(* Logix 5000 project; controller SX_V040001_C001 vendor 1 type 14 code 77 rev 16.22; software revision 16.04; part 33 of 35 *)
(* tags used below, declared in another part *)
   ALL_KINDS : INT[90];
   CMD : INT[36];
   EMPTYING : INT[18];
   G_DInput : DINT[3];
   loading : INT[19];
   METERING : INT[44];
   PARAMETER : INT[501];
   RECIPE_GENERAL : INT[405];
   REMOTE_DATA_IN : INT[510];
   REMOTE_DATA_OUT : INT[510];
   REMOTE_RECIPE : INT[405];
   REMOTE_SYSTEM : INT[38];
   RM_CMD : INT[9];
   s_bcc : INT;
   STATUS_SEND_PART_1 : INT[135];
   T_LIVEBIT_OFF : TIMER;
   T_LIVEBIT_ON : TIMER;
(* MainProgram, continued *)

ROUTINE RemoteComDeco_Direct   (* ladder *)
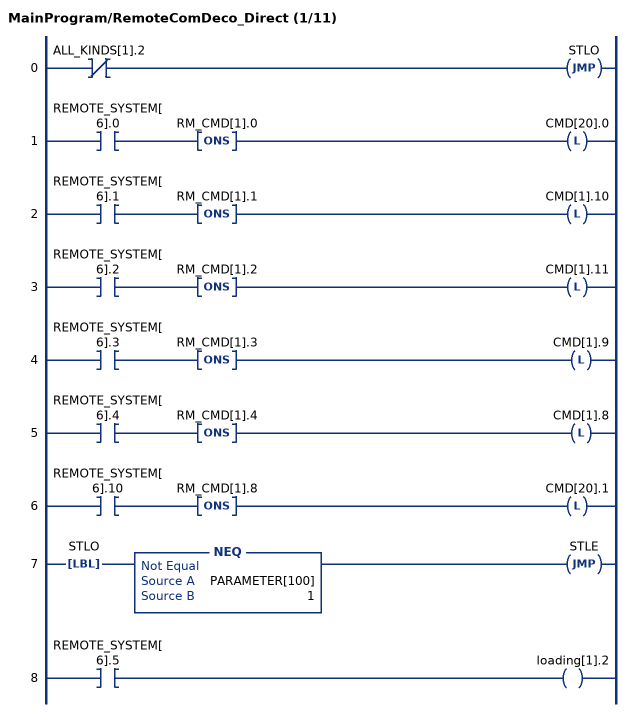
   0: XIO(ALL_KINDS[1].2)JMP(STLO);
   1: XIC(REMOTE_SYSTEM[6].0)ONS(RM_CMD[1].0)OTL(CMD[20].0);
   2: XIC(REMOTE_SYSTEM[6].1)ONS(RM_CMD[1].1)OTL(CMD[1].10);
   3: XIC(REMOTE_SYSTEM[6].2)ONS(RM_CMD[1].2)OTL(CMD[1].11);
   4: XIC(REMOTE_SYSTEM[6].3)ONS(RM_CMD[1].3)OTL(CMD[1].9);
   5: XIC(REMOTE_SYSTEM[6].4)ONS(RM_CMD[1].4)OTL(CMD[1].8);
   6: XIC(REMOTE_SYSTEM[6].10)ONS(RM_CMD[1].8)OTL(CMD[20].1);
   7: LBL(STLO)NEQ(PARAMETER[100],1)JMP(STLE);
   8: XIC(REMOTE_SYSTEM[6].5)OTE(loading[1].2);
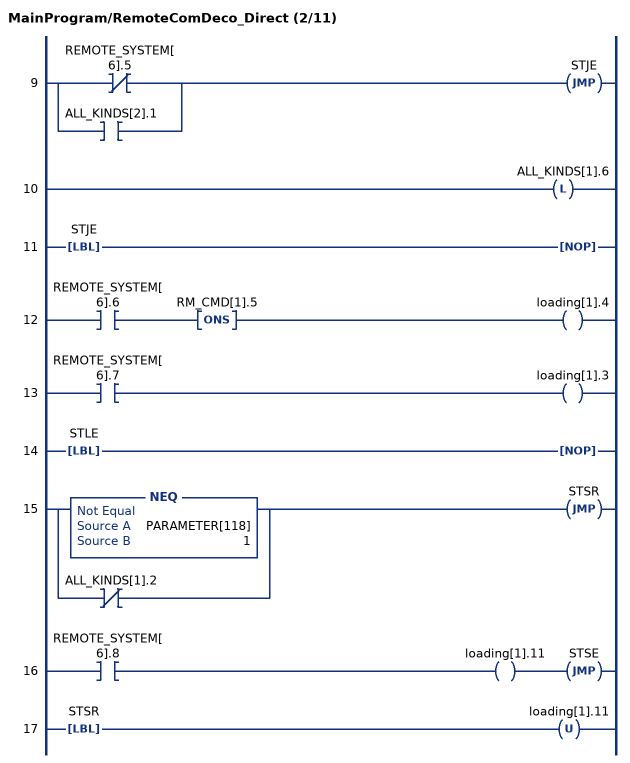
   9: [XIO(REMOTE_SYSTEM[6].5) ,XIC(ALL_KINDS[2].1) ]JMP(STJE);
   10: OTL(ALL_KINDS[1].6);
   11: LBL(STJE)NOP();
   12: XIC(REMOTE_SYSTEM[6].6)ONS(RM_CMD[1].5)OTE(loading[1].4);
   13: XIC(REMOTE_SYSTEM[6].7)OTE(loading[1].3);
   14: LBL(STLE)NOP();
   15: [NEQ(PARAMETER[118],1) ,XIO(ALL_KINDS[1].2) ]JMP(STSR);
   16: XIC(REMOTE_SYSTEM[6].8)OTE(loading[1].11)JMP(STSE);
   17: LBL(STSR)OTU(loading[1].11);
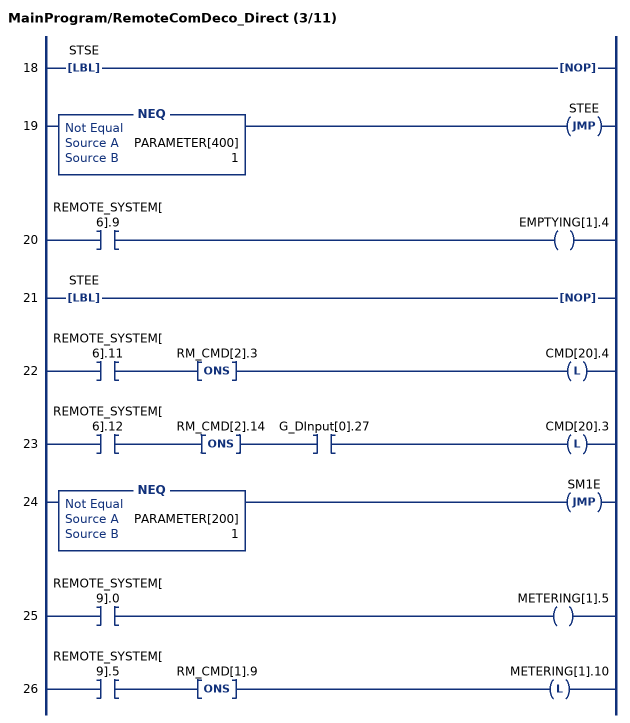
   18: LBL(STSE)NOP();
   19: NEQ(PARAMETER[400],1)JMP(STEE);
   20: XIC(REMOTE_SYSTEM[6].9)OTE(EMPTYING[1].4);
   21: LBL(STEE)NOP();
   22: XIC(REMOTE_SYSTEM[6].11)ONS(RM_CMD[2].3)OTL(CMD[20].4);
   23: XIC(REMOTE_SYSTEM[6].12)ONS(RM_CMD[2].14)XIC(G_DInput[0].27)OTL(CMD[20].3);
   24: NEQ(PARAMETER[200],1)JMP(SM1E);
   25: XIC(REMOTE_SYSTEM[9].0)OTE(METERING[1].5);
   26: XIC(REMOTE_SYSTEM[9].5)ONS(RM_CMD[1].9)OTL(METERING[1].10);
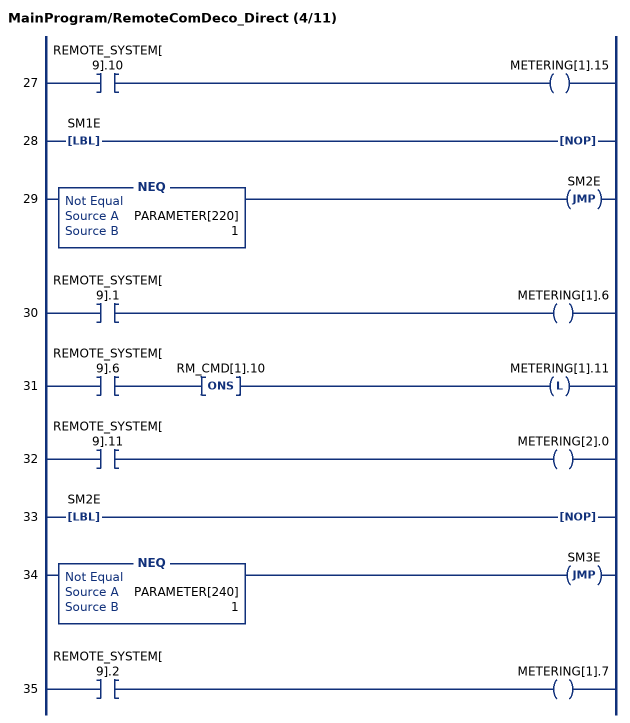
   27: XIC(REMOTE_SYSTEM[9].10)OTE(METERING[1].15);
   28: LBL(SM1E)NOP();
   29: NEQ(PARAMETER[220],1)JMP(SM2E);
   30: XIC(REMOTE_SYSTEM[9].1)OTE(METERING[1].6);
   31: XIC(REMOTE_SYSTEM[9].6)ONS(RM_CMD[1].10)OTL(METERING[1].11);
   32: XIC(REMOTE_SYSTEM[9].11)OTE(METERING[2].0);
   33: LBL(SM2E)NOP();
   34: NEQ(PARAMETER[240],1)JMP(SM3E);
   35: XIC(REMOTE_SYSTEM[9].2)OTE(METERING[1].7);
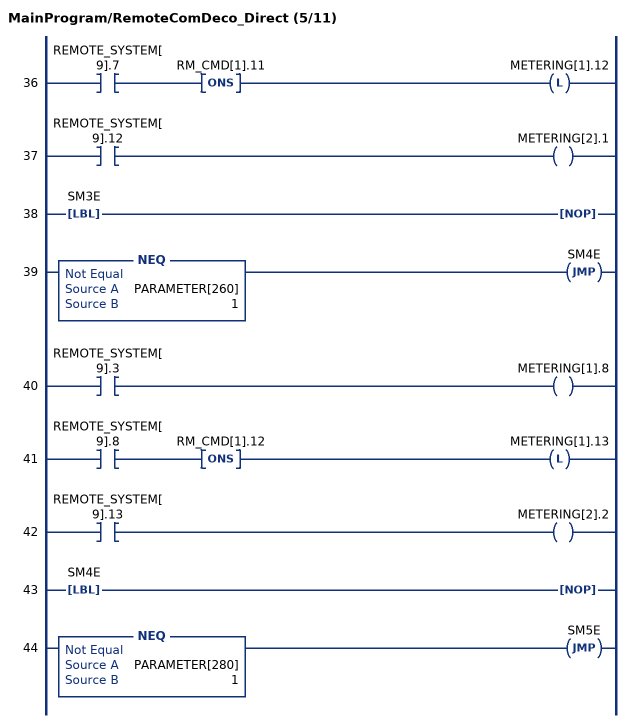
   36: XIC(REMOTE_SYSTEM[9].7)ONS(RM_CMD[1].11)OTL(METERING[1].12);
   37: XIC(REMOTE_SYSTEM[9].12)OTE(METERING[2].1);
   38: LBL(SM3E)NOP();
   39: NEQ(PARAMETER[260],1)JMP(SM4E);
   40: XIC(REMOTE_SYSTEM[9].3)OTE(METERING[1].8);
   41: XIC(REMOTE_SYSTEM[9].8)ONS(RM_CMD[1].12)OTL(METERING[1].13);
   42: XIC(REMOTE_SYSTEM[9].13)OTE(METERING[2].2);
   43: LBL(SM4E)NOP();
   44: NEQ(PARAMETER[280],1)JMP(SM5E);
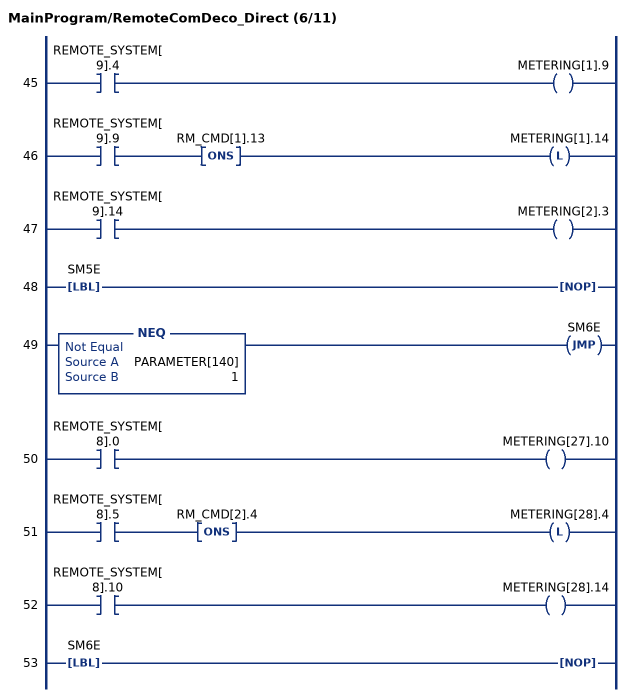
   45: XIC(REMOTE_SYSTEM[9].4)OTE(METERING[1].9);
   46: XIC(REMOTE_SYSTEM[9].9)ONS(RM_CMD[1].13)OTL(METERING[1].14);
   47: XIC(REMOTE_SYSTEM[9].14)OTE(METERING[2].3);
   48: LBL(SM5E)NOP();
   49: NEQ(PARAMETER[140],1)JMP(SM6E);
   50: XIC(REMOTE_SYSTEM[8].0)OTE(METERING[27].10);
   51: XIC(REMOTE_SYSTEM[8].5)ONS(RM_CMD[2].4)OTL(METERING[28].4);
   52: XIC(REMOTE_SYSTEM[8].10)OTE(METERING[28].14);
   53: LBL(SM6E)NOP();
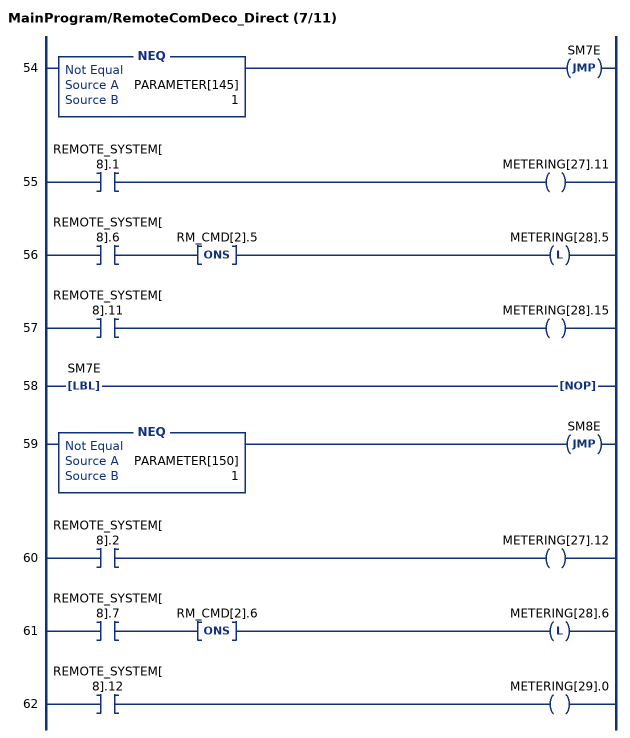
   54: NEQ(PARAMETER[145],1)JMP(SM7E);
   55: XIC(REMOTE_SYSTEM[8].1)OTE(METERING[27].11);
   56: XIC(REMOTE_SYSTEM[8].6)ONS(RM_CMD[2].5)OTL(METERING[28].5);
   57: XIC(REMOTE_SYSTEM[8].11)OTE(METERING[28].15);
   58: LBL(SM7E)NOP();
   59: NEQ(PARAMETER[150],1)JMP(SM8E);
   60: XIC(REMOTE_SYSTEM[8].2)OTE(METERING[27].12);
   61: XIC(REMOTE_SYSTEM[8].7)ONS(RM_CMD[2].6)OTL(METERING[28].6);
   62: XIC(REMOTE_SYSTEM[8].12)OTE(METERING[29].0);
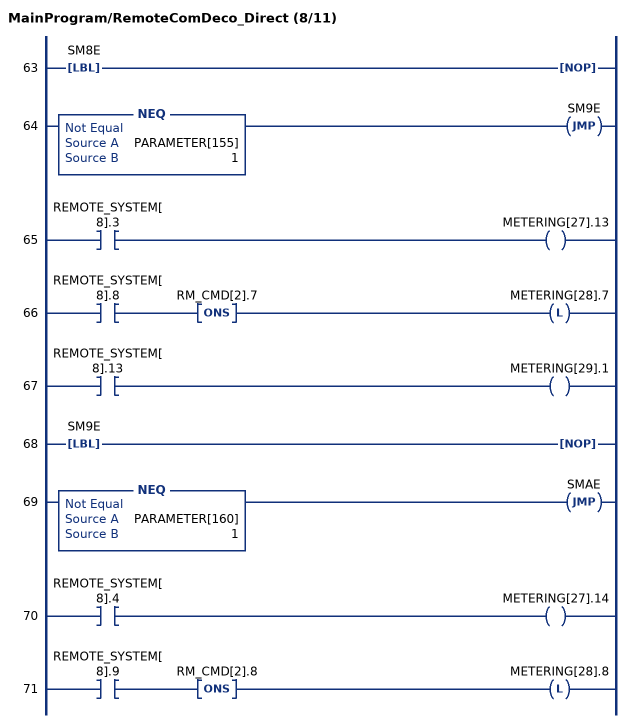
   63: LBL(SM8E)NOP();
   64: NEQ(PARAMETER[155],1)JMP(SM9E);
   65: XIC(REMOTE_SYSTEM[8].3)OTE(METERING[27].13);
   66: XIC(REMOTE_SYSTEM[8].8)ONS(RM_CMD[2].7)OTL(METERING[28].7);
   67: XIC(REMOTE_SYSTEM[8].13)OTE(METERING[29].1);
   68: LBL(SM9E)NOP();
   69: NEQ(PARAMETER[160],1)JMP(SMAE);
   70: XIC(REMOTE_SYSTEM[8].4)OTE(METERING[27].14);
   71: XIC(REMOTE_SYSTEM[8].9)ONS(RM_CMD[2].8)OTL(METERING[28].8);
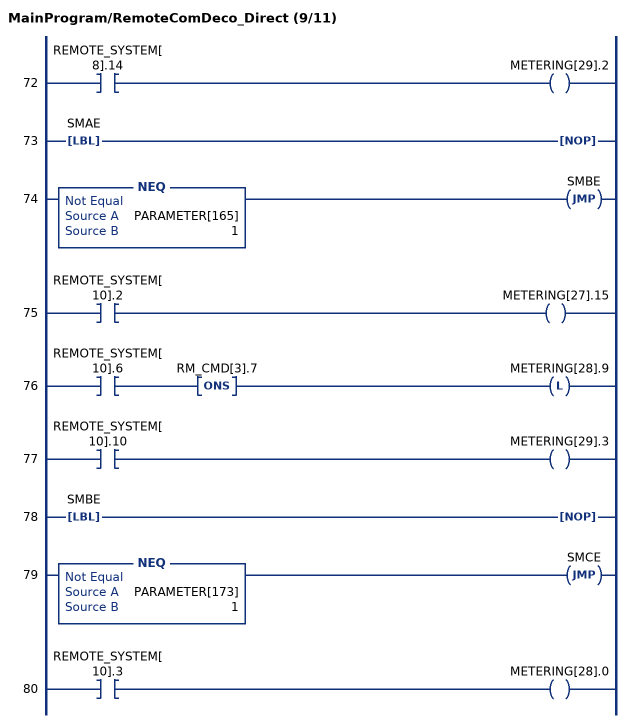
   72: XIC(REMOTE_SYSTEM[8].14)OTE(METERING[29].2);
   73: LBL(SMAE)NOP();
   74: NEQ(PARAMETER[165],1)JMP(SMBE);
   75: XIC(REMOTE_SYSTEM[10].2)OTE(METERING[27].15);
   76: XIC(REMOTE_SYSTEM[10].6)ONS(RM_CMD[3].7)OTL(METERING[28].9);
   77: XIC(REMOTE_SYSTEM[10].10)OTE(METERING[29].3);
   78: LBL(SMBE)NOP();
   79: NEQ(PARAMETER[173],1)JMP(SMCE);
   80: XIC(REMOTE_SYSTEM[10].3)OTE(METERING[28].0);
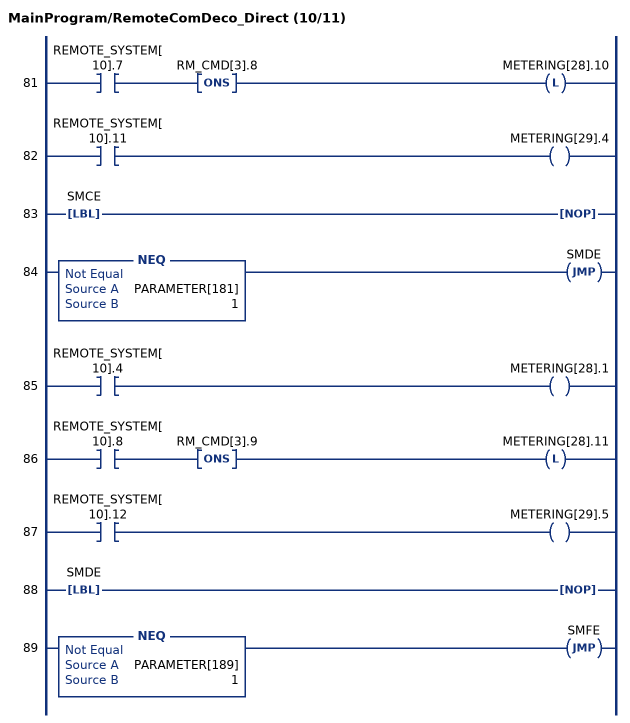
   81: XIC(REMOTE_SYSTEM[10].7)ONS(RM_CMD[3].8)OTL(METERING[28].10);
   82: XIC(REMOTE_SYSTEM[10].11)OTE(METERING[29].4);
   83: LBL(SMCE)NOP();
   84: NEQ(PARAMETER[181],1)JMP(SMDE);
   85: XIC(REMOTE_SYSTEM[10].4)OTE(METERING[28].1);
   86: XIC(REMOTE_SYSTEM[10].8)ONS(RM_CMD[3].9)OTL(METERING[28].11);
   87: XIC(REMOTE_SYSTEM[10].12)OTE(METERING[29].5);
   88: LBL(SMDE)NOP();
   89: NEQ(PARAMETER[189],1)JMP(SMFE);
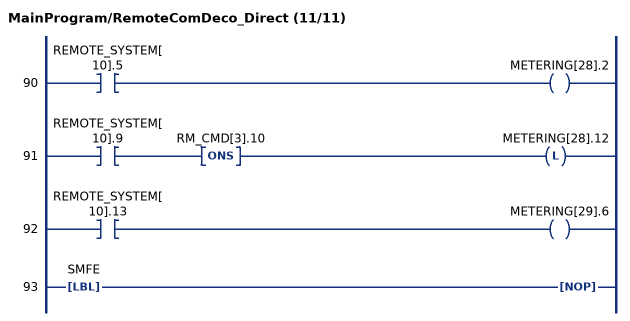
   90: XIC(REMOTE_SYSTEM[10].5)OTE(METERING[28].2);
   91: XIC(REMOTE_SYSTEM[10].9)ONS(RM_CMD[3].10)OTL(METERING[28].12);
   92: XIC(REMOTE_SYSTEM[10].13)OTE(METERING[29].6);
   93: LBL(SMFE)NOP();
END_ROUTINE

ROUTINE RemoteSystemHandler   (* ladder *)
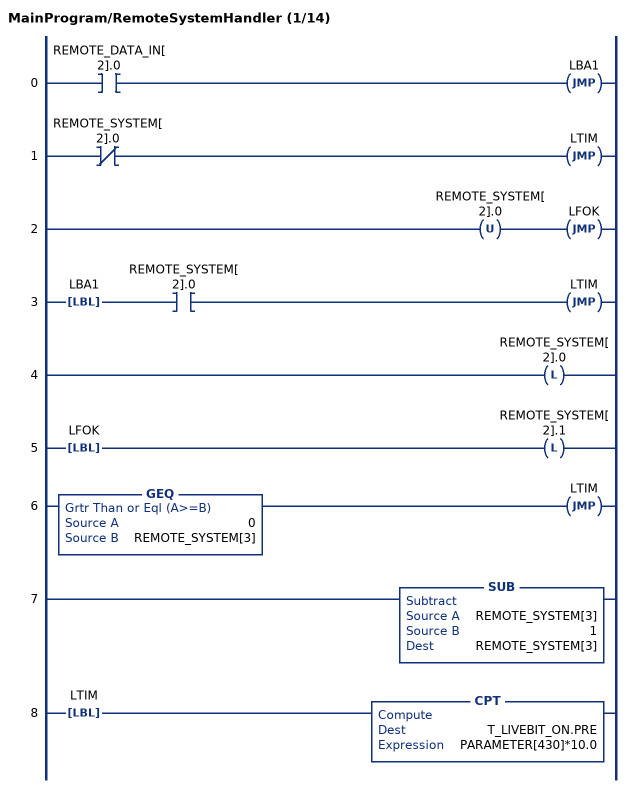
   0: XIC(REMOTE_DATA_IN[2].0)JMP(LBA1);
   1: XIO(REMOTE_SYSTEM[2].0)JMP(LTIM);
   2: OTU(REMOTE_SYSTEM[2].0)JMP(LFOK);
   3: LBL(LBA1)XIC(REMOTE_SYSTEM[2].0)JMP(LTIM);
   4: OTL(REMOTE_SYSTEM[2].0);
   5: LBL(LFOK)OTL(REMOTE_SYSTEM[2].1);
   6: GEQ(0,REMOTE_SYSTEM[3])JMP(LTIM);
   7: SUB(REMOTE_SYSTEM[3],1,REMOTE_SYSTEM[3]);
   8: LBL(LTIM)CPT(T_LIVEBIT_ON.PRE,PARAMETER[430]*10.0);
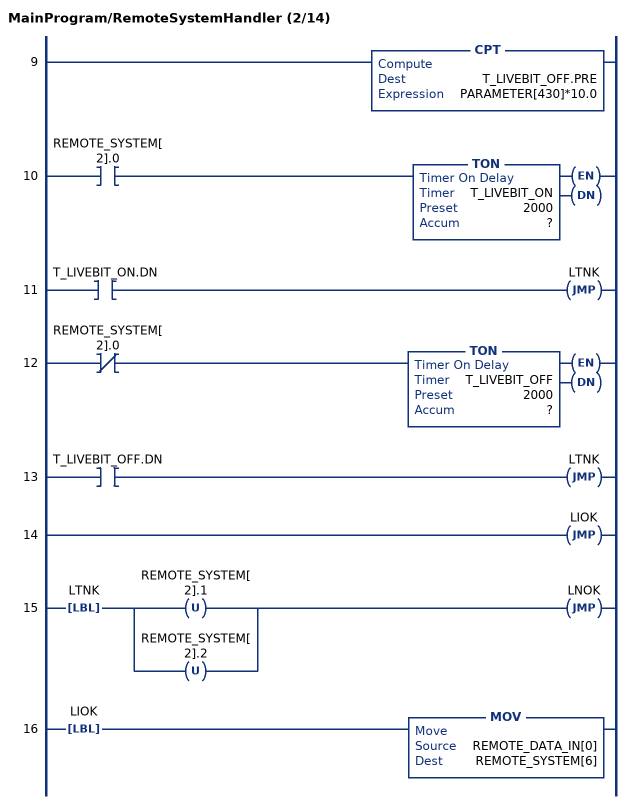
   9: CPT(T_LIVEBIT_OFF.PRE,PARAMETER[430]*10.0);
   10: XIC(REMOTE_SYSTEM[2].0)TON(T_LIVEBIT_ON,?,?);
   11: XIC(T_LIVEBIT_ON.DN)JMP(LTNK);
   12: XIO(REMOTE_SYSTEM[2].0)TON(T_LIVEBIT_OFF,?,?);
   13: XIC(T_LIVEBIT_OFF.DN)JMP(LTNK);
   14: JMP(LIOK);
   15: LBL(LTNK)[OTU(REMOTE_SYSTEM[2].1) ,OTU(REMOTE_SYSTEM[2].2) ]JMP(LNOK);
   16: LBL(LIOK)MOV(REMOTE_DATA_IN[0],REMOTE_SYSTEM[6]);
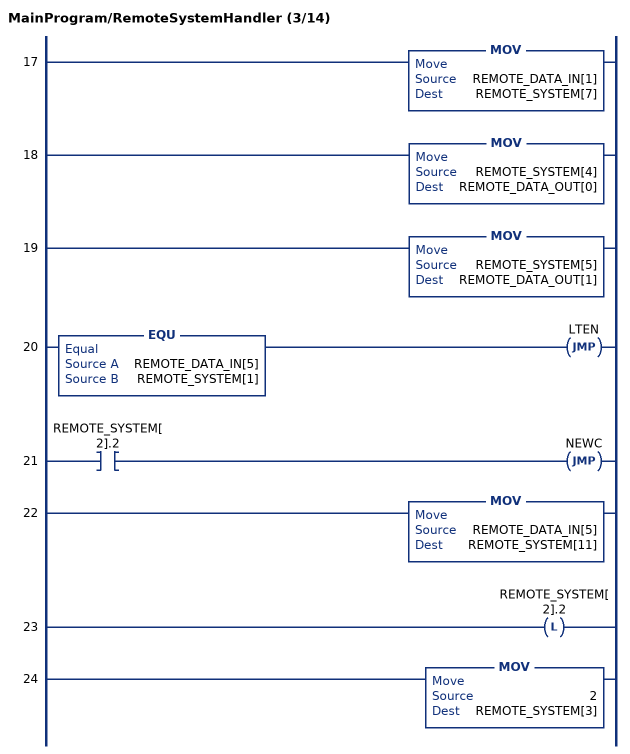
   17: MOV(REMOTE_DATA_IN[1],REMOTE_SYSTEM[7]);
   18: MOV(REMOTE_SYSTEM[4],REMOTE_DATA_OUT[0]);
   19: MOV(REMOTE_SYSTEM[5],REMOTE_DATA_OUT[1]);
   20: EQU(REMOTE_DATA_IN[5],REMOTE_SYSTEM[1])JMP(LTEN);
   21: XIC(REMOTE_SYSTEM[2].2)JMP(NEWC);
   22: MOV(REMOTE_DATA_IN[5],REMOTE_SYSTEM[11]);
   23: OTL(REMOTE_SYSTEM[2].2);
   24: MOV(2,REMOTE_SYSTEM[3]);
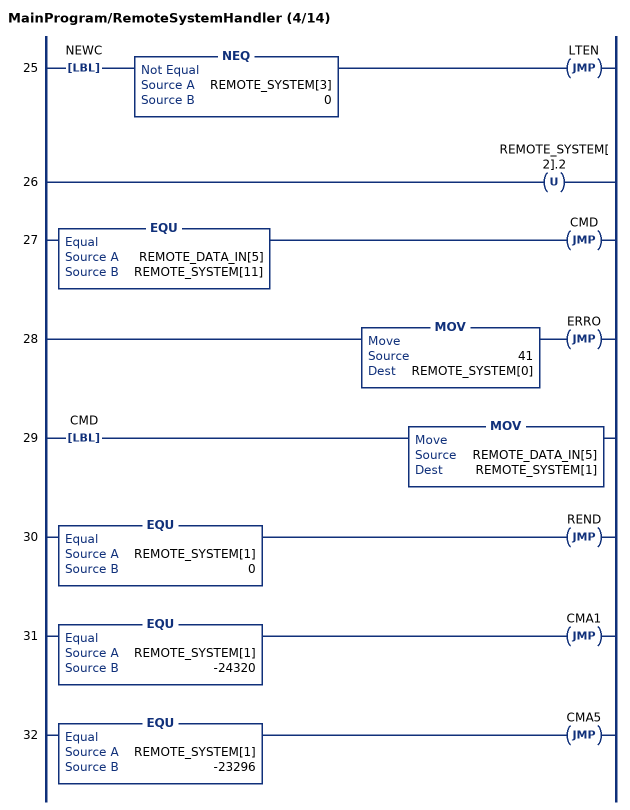
   25: LBL(NEWC)NEQ(REMOTE_SYSTEM[3],0)JMP(LTEN);
   26: OTU(REMOTE_SYSTEM[2].2);
   27: EQU(REMOTE_DATA_IN[5],REMOTE_SYSTEM[11])JMP(CMD);
   28: MOV(41,REMOTE_SYSTEM[0])JMP(ERRO);
   29: LBL(CMD)MOV(REMOTE_DATA_IN[5],REMOTE_SYSTEM[1]);
   30: EQU(REMOTE_SYSTEM[1],0)JMP(REND);
   31: EQU(REMOTE_SYSTEM[1],-24320)JMP(CMA1);
   32: EQU(REMOTE_SYSTEM[1],-23296)JMP(CMA5);
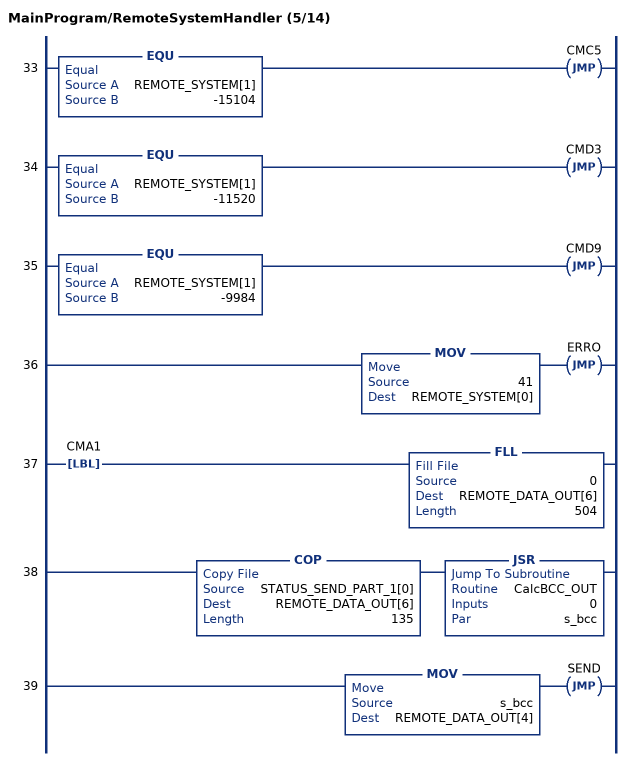
   33: EQU(REMOTE_SYSTEM[1],-15104)JMP(CMC5);
   34: EQU(REMOTE_SYSTEM[1],-11520)JMP(CMD3);
   35: EQU(REMOTE_SYSTEM[1],-9984)JMP(CMD9);
   36: MOV(41,REMOTE_SYSTEM[0])JMP(ERRO);
   37: LBL(CMA1)FLL(0,REMOTE_DATA_OUT[6],504);
   38: COP(STATUS_SEND_PART_1[0],REMOTE_DATA_OUT[6],135)JSR(CalcBCC_OUT,0,s_bcc);
   39: MOV(s_bcc,REMOTE_DATA_OUT[4])JMP(SEND);
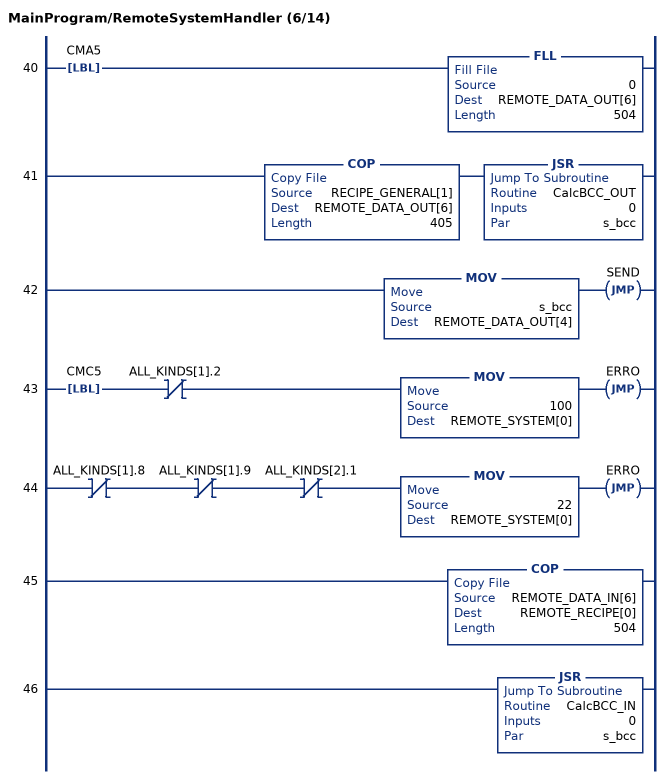
   40: LBL(CMA5)FLL(0,REMOTE_DATA_OUT[6],504);
   41: COP(RECIPE_GENERAL[1],REMOTE_DATA_OUT[6],405)JSR(CalcBCC_OUT,0,s_bcc);
   42: MOV(s_bcc,REMOTE_DATA_OUT[4])JMP(SEND);
   43: LBL(CMC5)XIO(ALL_KINDS[1].2)MOV(100,REMOTE_SYSTEM[0])JMP(ERRO);
   44: XIO(ALL_KINDS[1].8)XIO(ALL_KINDS[1].9)XIO(ALL_KINDS[2].1)MOV(22,REMOTE_SYSTEM[0])JMP(ERRO);
   45: COP(REMOTE_DATA_IN[6],REMOTE_RECIPE[0],504);
   46: JSR(CalcBCC_IN,0,s_bcc);
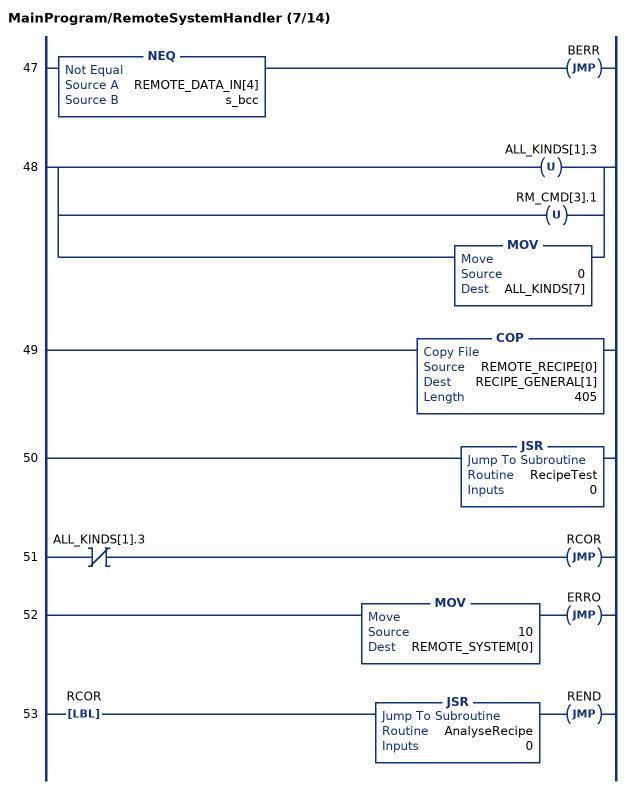
   47: NEQ(REMOTE_DATA_IN[4],s_bcc)JMP(BERR);
   48: [OTU(ALL_KINDS[1].3) ,OTU(RM_CMD[3].1) ,MOV(0,ALL_KINDS[7]) ];
   49: COP(REMOTE_RECIPE[0],RECIPE_GENERAL[1],405);
   50: JSR(RecipeTest,0);
   51: XIO(ALL_KINDS[1].3)JMP(RCOR);
   52: MOV(10,REMOTE_SYSTEM[0])JMP(ERRO);
   53: LBL(RCOR)JSR(AnalyseRecipe,0)JMP(REND);
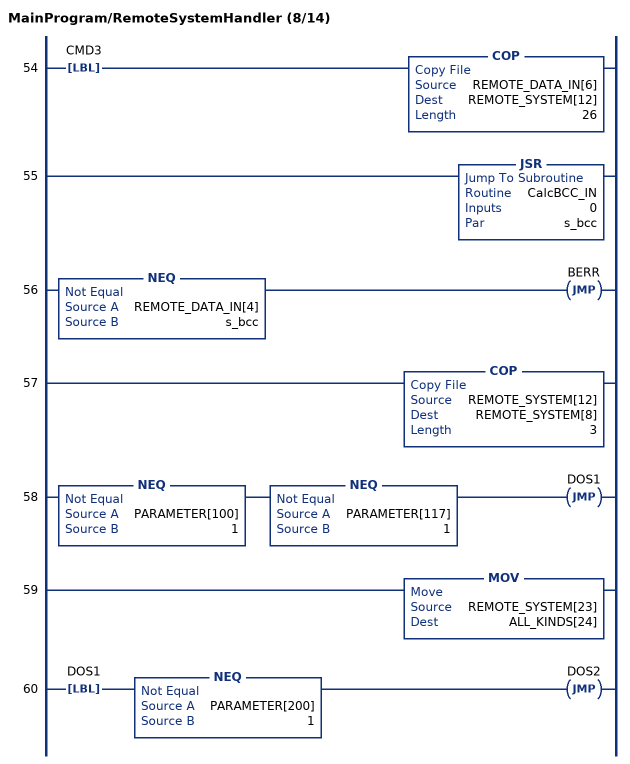
   54: LBL(CMD3)COP(REMOTE_DATA_IN[6],REMOTE_SYSTEM[12],26);
   55: JSR(CalcBCC_IN,0,s_bcc);
   56: NEQ(REMOTE_DATA_IN[4],s_bcc)JMP(BERR);
   57: COP(REMOTE_SYSTEM[12],REMOTE_SYSTEM[8],3);
   58: NEQ(PARAMETER[100],1)NEQ(PARAMETER[117],1)JMP(DOS1);
   59: MOV(REMOTE_SYSTEM[23],ALL_KINDS[24]);
   60: LBL(DOS1)NEQ(PARAMETER[200],1)JMP(DOS2);
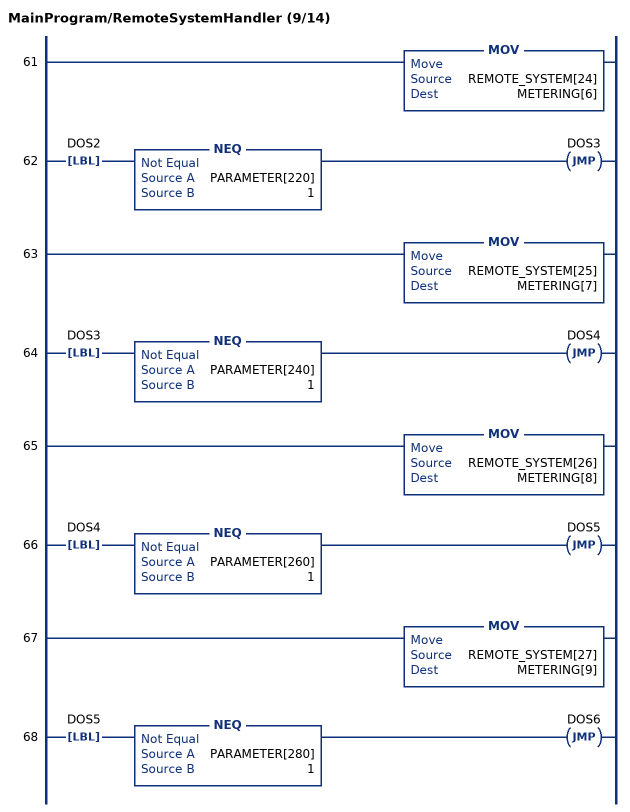
   61: MOV(REMOTE_SYSTEM[24],METERING[6]);
   62: LBL(DOS2)NEQ(PARAMETER[220],1)JMP(DOS3);
   63: MOV(REMOTE_SYSTEM[25],METERING[7]);
   64: LBL(DOS3)NEQ(PARAMETER[240],1)JMP(DOS4);
   65: MOV(REMOTE_SYSTEM[26],METERING[8]);
   66: LBL(DOS4)NEQ(PARAMETER[260],1)JMP(DOS5);
   67: MOV(REMOTE_SYSTEM[27],METERING[9]);
   68: LBL(DOS5)NEQ(PARAMETER[280],1)JMP(DOS6);
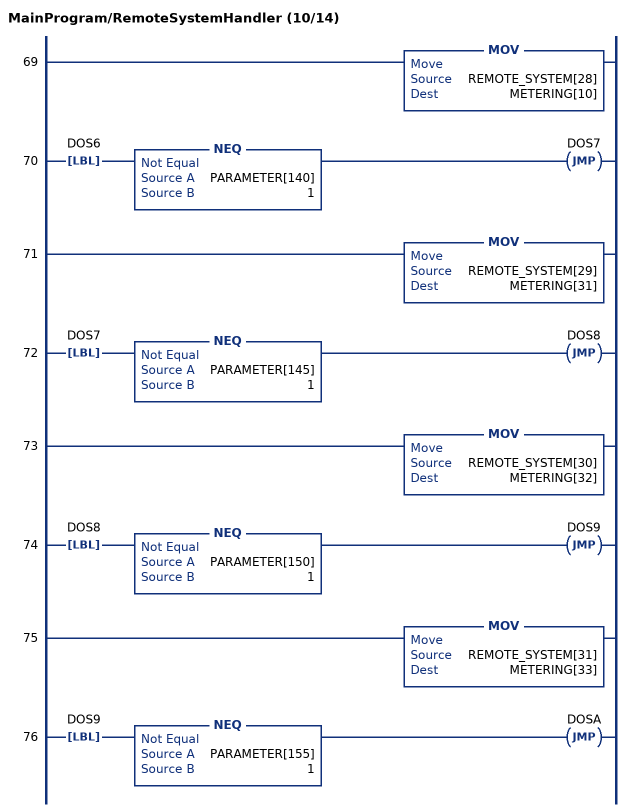
   69: MOV(REMOTE_SYSTEM[28],METERING[10]);
   70: LBL(DOS6)NEQ(PARAMETER[140],1)JMP(DOS7);
   71: MOV(REMOTE_SYSTEM[29],METERING[31]);
   72: LBL(DOS7)NEQ(PARAMETER[145],1)JMP(DOS8);
   73: MOV(REMOTE_SYSTEM[30],METERING[32]);
   74: LBL(DOS8)NEQ(PARAMETER[150],1)JMP(DOS9);
   75: MOV(REMOTE_SYSTEM[31],METERING[33]);
   76: LBL(DOS9)NEQ(PARAMETER[155],1)JMP(DOSA);
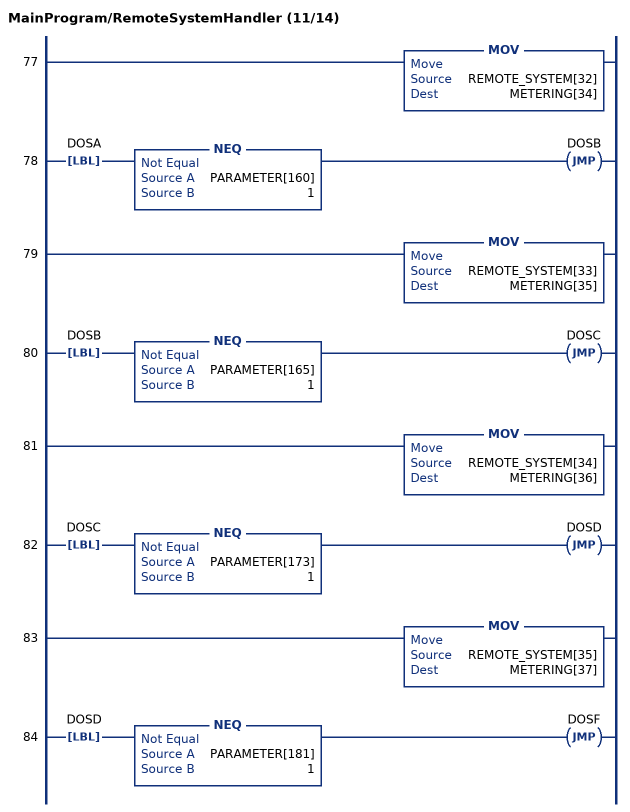
   77: MOV(REMOTE_SYSTEM[32],METERING[34]);
   78: LBL(DOSA)NEQ(PARAMETER[160],1)JMP(DOSB);
   79: MOV(REMOTE_SYSTEM[33],METERING[35]);
   80: LBL(DOSB)NEQ(PARAMETER[165],1)JMP(DOSC);
   81: MOV(REMOTE_SYSTEM[34],METERING[36]);
   82: LBL(DOSC)NEQ(PARAMETER[173],1)JMP(DOSD);
   83: MOV(REMOTE_SYSTEM[35],METERING[37]);
   84: LBL(DOSD)NEQ(PARAMETER[181],1)JMP(DOSF);
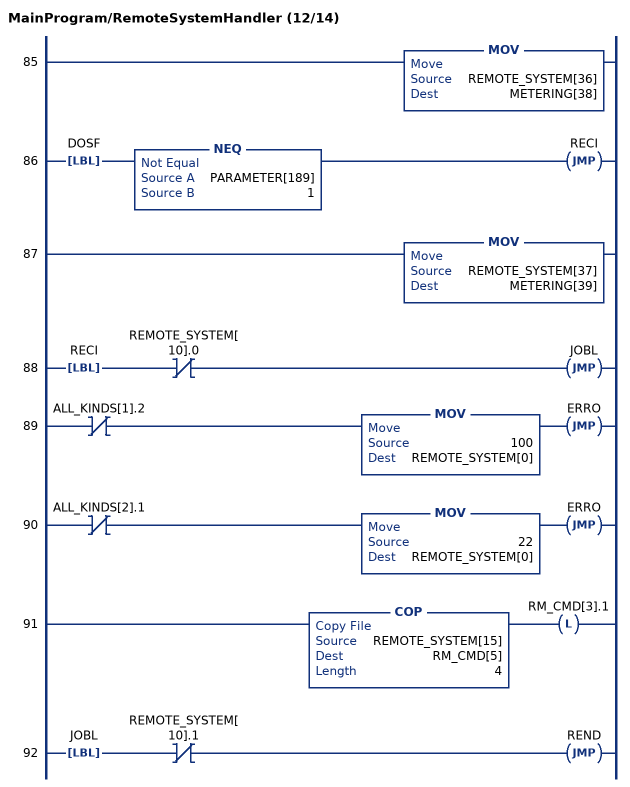
   85: MOV(REMOTE_SYSTEM[36],METERING[38]);
   86: LBL(DOSF)NEQ(PARAMETER[189],1)JMP(RECI);
   87: MOV(REMOTE_SYSTEM[37],METERING[39]);
   88: LBL(RECI)XIO(REMOTE_SYSTEM[10].0)JMP(JOBL);
   89: XIO(ALL_KINDS[1].2)MOV(100,REMOTE_SYSTEM[0])JMP(ERRO);
   90: XIO(ALL_KINDS[2].1)MOV(22,REMOTE_SYSTEM[0])JMP(ERRO);
   91: COP(REMOTE_SYSTEM[15],RM_CMD[5],4)OTL(RM_CMD[3].1);
   92: LBL(JOBL)XIO(REMOTE_SYSTEM[10].1)JMP(REND);
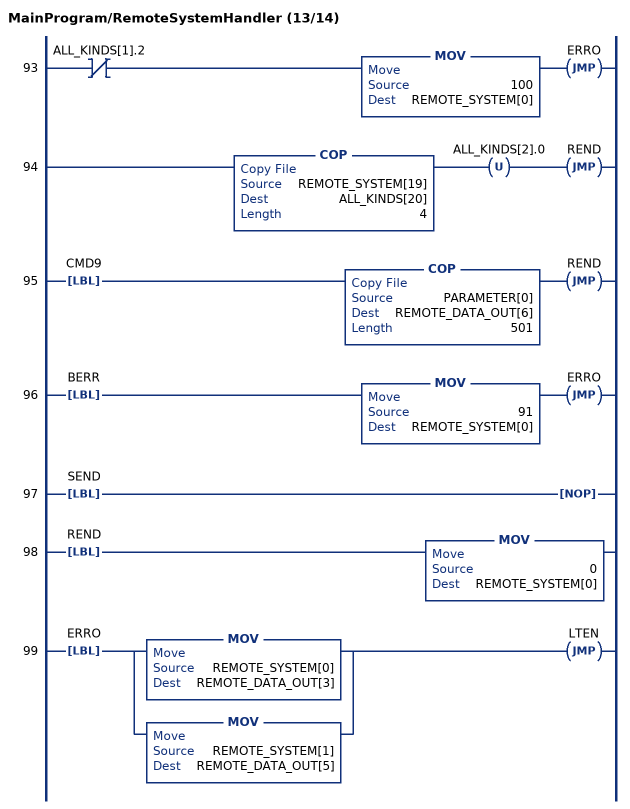
   93: XIO(ALL_KINDS[1].2)MOV(100,REMOTE_SYSTEM[0])JMP(ERRO);
   94: COP(REMOTE_SYSTEM[19],ALL_KINDS[20],4)OTU(ALL_KINDS[2].0)JMP(REND);
   95: LBL(CMD9)COP(PARAMETER[0],REMOTE_DATA_OUT[6],501)JMP(REND);
   96: LBL(BERR)MOV(91,REMOTE_SYSTEM[0])JMP(ERRO);
   97: LBL(SEND)NOP();
   98: LBL(REND)MOV(0,REMOTE_SYSTEM[0]);
   99: LBL(ERRO)[MOV(REMOTE_SYSTEM[0],REMOTE_DATA_OUT[3]) ,MOV(REMOTE_SYSTEM[1],REMOTE_DATA_OUT[5]) ]JMP(LTEN);
